KUKA KRL program: wartung.src, wartung.dat

--- wartung.src ---
&ACCESS RVO1
&REL 25
&COMMENT MANUTENCAO
&USER thsc160
&PARAM DISKPATH = KRC:\R1\Program
&PARAM version = 0.1
DEF wartung( )
;FOLD INI
  ;FOLD BASISTECH INI
    GLOBAL INTERRUPT DECL 3 WHEN $STOPMESS==TRUE DO IR_STOPM ( )
    BAS (#INITMOV,0 )
  ;ENDFOLD (BASISTECH INI)
;FOLD SPOTTECH INI
USERSPOT(#INIT)
;ENDFOLD (SPOTTECH INI)
;FOLD GRIPPERTECH INI
USER_GRP(0,DUMMY,DUMMY,GDEFAULT)
;ENDFOLD (GRIPPERTECH INI)
;FOLD USER INI

;Make your modifications here
;FOLD COLLISION_V_3.01 INI ;%{E}
    IF (COLLISION_DATA[1].I_NR>0) THEN
    GLOBAL INTERRUPT DECL 21 WHEN $IN[COLLISION_DATA[1].I_NR]==FALSE DO COLLSTOP (1,0 )
    ENDIF
    IF (COLLISION_DATA[2].I_NR>0) THEN
    GLOBAL INTERRUPT DECL 22 WHEN $IN[COLLISION_DATA[2].I_NR]==FALSE DO COLLSTOP (2,0 )
    ENDIF
    IF (COLLISION_DATA[3].I_NR>0) THEN
    GLOBAL INTERRUPT DECL 23 WHEN $IN[COLLISION_DATA[3].I_NR]==FALSE DO COLLSTOP (3,0 )
    ENDIF
    IF (COLLISION_DATA[4].I_NR>0) THEN
    GLOBAL INTERRUPT DECL 24 WHEN $IN[COLLISION_DATA[4].I_NR]==FALSE DO COLLSTOP (4,0 )
    ENDIF
;ENDFOLD (Collision)

;ENDFOLD (USER INI)

;ENDFOLD (INI)

;FOLD ; ESTACAO P13060;%{PE}%R 8.2.20,%MKUKATPBASIS,%CCOMMENT,%VNORMAL,%P 2:ESTACAO  P13060
;ENDFOLD
;FOLD ; ROBO 5;%{PE}%R 8.2.20,%MKUKATPBASIS,%CCOMMENT,%VNORMAL,%P 2:ROBO  5
;ENDFOLD
;FOLD ; PROGRAMA DE MANUTENCAO;%{PE}%R 8.2.20,%MKUKATPBASIS,%CCOMMENT,%VNORMAL,%P 2:PROGRAMA  DE  MANUTENCAO
;ENDFOLD

; Caracterização dos meios de produção: P13.060-R5
; Versão atual: 17/07/2013 Nome: Manutenção
; Change: C2

;FOLD PTP HOME Vel=100 % DEFAULT;%{PE}%R 8.2.20,%MKUKATPBASIS,%CMOVE,%VPTP,%P 1:PTP, 2:HOME, 3:, 5:100, 7:DEFAULT
$BWDSTART=FALSE
PDAT_ACT=PDEFAULT
FDAT_ACT=FHOME
BAS(#PTP_PARAMS,100)
$H_POS=XHOME
PTP XHOME
;ENDFOLD

chk_w2_wechs_ok ()            ; check c1
wkz2_ab ()

;FOLD PTP HOME1 Vel=100 % DEFAULT;%{PE}%R 8.2.20,%MKUKATPBASIS,%CMOVE,%VPTP,%P 1:PTP, 2:HOME1, 3:, 5:100, 7:DEFAULT
$BWDSTART=FALSE
PDAT_ACT=PDEFAULT
FDAT_ACT=FHOME1
BAS(#PTP_PARAMS,100)
PTP XHOME1
;ENDFOLD

chk_w8_wechs_ok ()            ; check toolchanger
wkz3_an ()
chk_w3_wechs_ok ( )           ; VERIFICAÇÃO DE FERRAMENA: C2

;FOLD PTP Maintenance Vel=100 % PDAT10;%{PE}%R 8.2.20,%MKUKATPBASIS,%CMOVE,%VPTP,%P 1:PTP, 2:Maintenance, 3:, 5:100, 7:PDAT10
$BWDSTART=FALSE
PDAT_ACT=PPDAT10
FDAT_ACT=FMaintenance
BAS(#PTP_PARAMS,100)
PTP XMaintenance
;ENDFOLD

MSG_SHOW("DAI_H_Prog",#notify,999,"dai_maintenance_0")
;FOLD OUT 3218 'WPER:Wartungspos. erreicht'  State= TRUE ;%{PE}%R 5.2.22,%MKUKATPBASIS,%COUT,%VOUTX,%P 2:3218, 3:WPER:Wartungspos. erreicht, 5:TRUE, 6:
    $OUT[3218]=TRUE
;ENDFOLD
;FOLD WAIT FOR ( NOT IN 3218 'ANFWP:Anforderung Wartungspos.' );%{PE}%R 5.2.22,%MKUKATPBASIS,%CEXT_WAIT_FOR,%VEXT_WAIT_FOR,%P 2:, 4:NOT, 5:$IN, 6:3218, 7:ANFWP:Anforderung Wartungspos., 9:
    WAIT FOR  (  NOT $IN[3218] )
;ENDFOLD




;FOLD OUT 3218 'WPER:Wartungspos. erreicht'  State= FALSE ;%{PE}%R 5.2.22,%MKUKATPBASIS,%COUT,%VOUTX,%P 2:3218, 3:WPER:Wartungspos. erreicht, 5:FALSE, 6:
    $OUT[3218]=FALSE
;ENDFOLD

;FOLD PTP P1 PDAT7 SPOT Gun=2 RETR OPN PgNo1=1 ACTIVE=1 Tool[3]:Gun C2 Base[0];%{PE}%R 8.2.2,%MKUKATPSPOT,%CSPOT,%VPTP,%P 1:PTP, 2:P1, 3:, 5:100, 7:PDAT7, 10:2, 12:#FIRST, 14:#OPN, 16:1, 18:1, 20:0, 22:0, 24:1, 25:NORMAL
$BWDSTART=FALSE
PDAT_ACT=PPDAT7
FDAT_ACT=FP1
BAS(#PTP_PARAMS,PPDAT7.VEL)
S_ACT.GUN=2
S_ACT.PAIR=SDEFAULT.PAIR
S_ACT.RETR=#OPN
S_ACT.CLO_TM=1
S_ACT.PGNO1=1
S_ACT.PGNO2=SDEFAULT.PGNO2
S_ACT.PRESS1=SDEFAULT.PRESS1
S_ACT.PRESS2=SDEFAULT.PRESS2
S_READY=FALSE
PTP XP1
USERSPOT(#SPOT, S_ACT)
WAIT FOR S_READY
;ENDFOLD

;FOLD PTP HOME1 Vel=100 % DEFAULT;%{PE}%R 8.2.20,%MKUKATPBASIS,%CMOVE,%VPTP,%P 1:PTP, 2:HOME1, 3:, 5:100, 7:DEFAULT
$BWDSTART=FALSE
PDAT_ACT=PDEFAULT
FDAT_ACT=FHOME1
BAS(#PTP_PARAMS,100)
PTP XHOME1
;ENDFOLD

chk_w3_wechs_ok ()     ; check c2
wkz3_ab ()

;FOLD PTP HOME Vel=100 % DEFAULT;%{PE}%R 8.2.17,%MKUKATPBASIS,%CMOVE,%VPTP,%P 1:PTP, 2:HOME, 3:, 5:100, 7:DEFAULT
$BWDSTART=FALSE
PDAT_ACT=PDEFAULT
FDAT_ACT=FHOME
BAS(#PTP_PARAMS,100)
$H_POS=XHOME
PTP XHOME
;ENDFOLD

chk_w8_wechs_ok ()     ;check toolchanger
wkz2_an ()
chk_w2_wechs_ok ( )    ; VERIFICAÇÃO DE FERRAMENA: C1

END

--- wartung.dat ---
&ACCESS RVO1
&REL 25
&COMMENT MANUTENCAO
&USER thsc160
&PARAM DISKPATH = KRC:\R1\Program
&PARAM version = 0.1
DEFDAT  wartung
;FOLD EXTERNAL DECLARATIONS;%{PE}%MKUKATPBASIS,%CEXT,%VCOMMON,%P
;FOLD GRIPPERTECH EXT
EXT  H50 (INT  :IN,INT  :IN,INT  :IN,GRP_TYP  :IN )
;ENDFOLD (GRIPPERTECH EXT)
;FOLD SPOTTECH EXT
EXT  USERSPOT (S_COMMAND  :IN,SPOT_TYPE  :IN )
;ENDFOLD (SPOTTECH EXT)
;FOLD BASISTECH EXT;%{PE}%MKUKATPBASIS,%CEXT,%VEXT,%P
EXT  BAS (BAS_COMMAND  :IN,REAL  :IN )
DECL INT SUCCESS
;ENDFOLD (BASISTECH EXT)
;FOLD USER EXT;%{E}%MKUKATPUSER,%CEXT,%VEXT,%P
;Make here your modifications
;FOLD COLLISION
EXT  COLLSTOP (INT  :IN,INT  :IN )
;ENDFOLD  (Collision)
;ENDFOLD (USER EXT)
;ENDFOLD (EXTERNAL DECLERATIONS)



DECL FDAT FHOME={TOOL_NO 0,BASE_NO 0,IPO_FRAME #BASE}

DECL E6AXIS XMaintenance={A1 -156.938995,A2 -118.107498,A3 89.710083,A4 -6.04678917,A5 45.7215691,A6 202.632507,E1 0.0,E2 0.0,E3 0.0,E4 0.0,E5 0.0,E6 0.0}
DECL FDAT FMaintenance={TOOL_NO 3,BASE_NO 0,IPO_FRAME #BASE,POINT2[] " ",TQ_STATE FALSE}

DECL PDAT PPDAT10={VEL 100.0,ACC 100.0,APO_DIST 100.0}
DECL FDAT FHOME1={TOOL_NO 0,BASE_NO 0,IPO_FRAME #BASE,POINT2[] " ",TQ_STATE FALSE}
DECL SPOT_SUGG_T LAST_SPOT={GUN[] "2                       ",RETR_CMD[] "#OPN                    ",CHOISE[] "#FIRST                  ",CLO_TM[] "1                       ",PGNO1[] "252                     ",PRESS1[] "0                       ",PGNO2[] "1                       ",PRESS2[] "0                       ",SPOT_PARAMS[] "NORMAL                  "}
DECL PDAT PPDAT7={VEL 100.0,ACC 100.0,APO_DIST 100.0,APO_MODE #CDIS}
DECL E6POS XP1={X -2102.61694,Y 828.297485,Z 1384.02197,A 162.000702,B 2.12318897,C -1.97843695,S 2,T 11,E1 0.0,E2 0.0,E3 0.0,E4 0.0,E5 0.0,E6 0.0}
DECL FDAT FP1={TOOL_NO 3,BASE_NO 0,IPO_FRAME #BASE,POINT2[] " ",TQ_STATE FALSE}
ENDDAT
